# EPICS substitutions: CryoControlApp/Db/wcmp_StartStop.substitutions
file wcmp_StartStop.vdb
{
         pattern { PLC_NAME            , AREA     , LOCA , CMPNUM }
                 { PLC_CP$(CP)2_CR1$(C), CP$(CP)2 , 1$(C),   4    }
}
